(* Logix 5000 project; controller STAT 1756-L72 rev 20.12; software revision 20.04; part 25 of 34 *)
(* tags used below, declared in another part *)
   B3 : DINT[35];
   N7 : DINT[150];
   N9 : DINT[200];
   S : INT[164];
   T4 : TIMER[100];
   tempo_d_lvl_H_decL1 : TIMER;
   tempo_on_lvl_H_decL1 : TIMER;
(* LANCY, continued *)

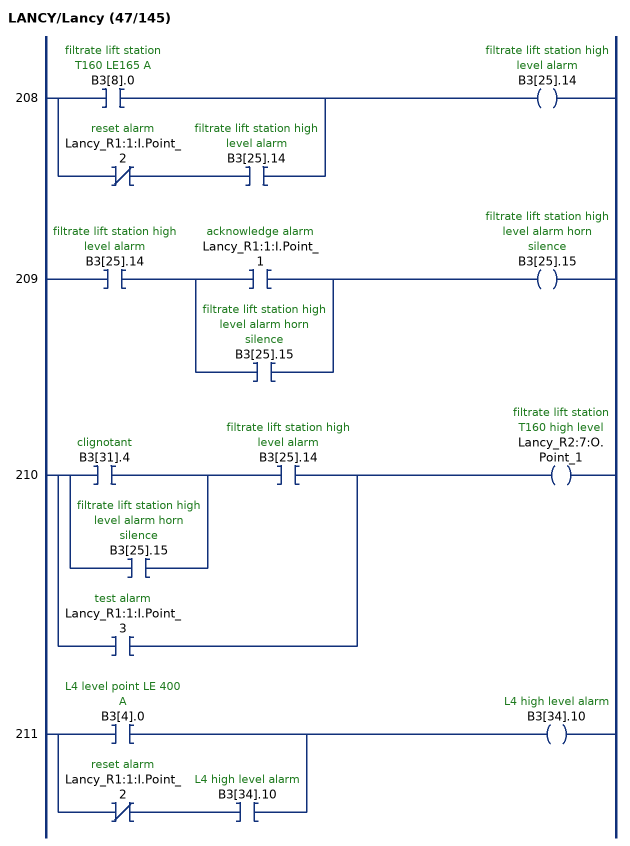
   208: [XIC(B3[8].0) ,XIO(Lancy_R1:1:I.Point_2) XIC(B3[25].14) ]OTE(B3[25].14);
   209: XIC(B3[25].14)[XIC(Lancy_R1:1:I.Point_1) ,XIC(B3[25].15) ]OTE(B3[25].15);
   210: [[XIC(B3[31].4) ,XIC(B3[25].15) ] XIC(B3[25].14) ,XIC(Lancy_R1:1:I.Point_3) ]OTE(Lancy_R2:7:O.Point_1);
   211: [XIC(B3[4].0) ,XIO(Lancy_R1:1:I.Point_2) XIC(B3[34].10) ]OTE(B3[34].10);
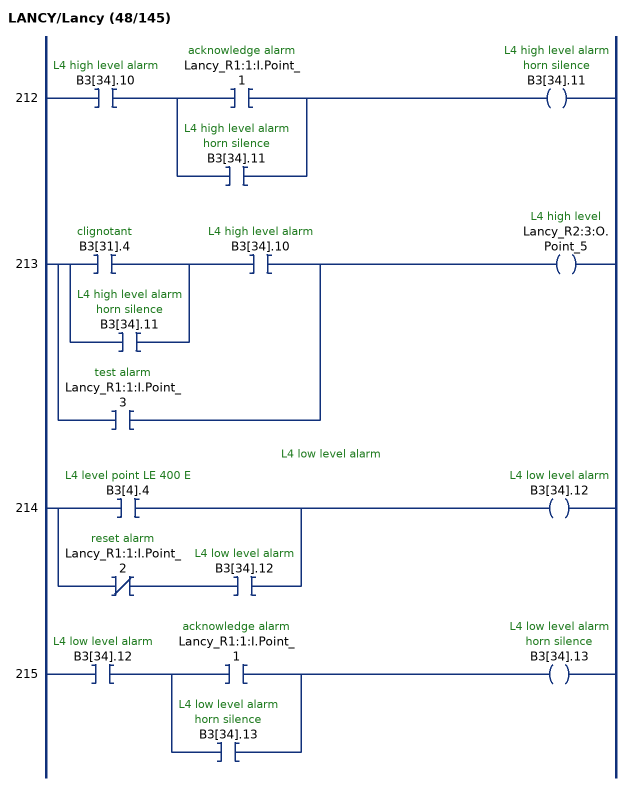
   212: XIC(B3[34].10)[XIC(Lancy_R1:1:I.Point_1) ,XIC(B3[34].11) ]OTE(B3[34].11);
   213: [[XIC(B3[31].4) ,XIC(B3[34].11) ] XIC(B3[34].10) ,XIC(Lancy_R1:1:I.Point_3) ]OTE(Lancy_R2:3:O.Point_5);
   // L4 low level alarm
   214: [XIC(B3[4].4) ,XIO(Lancy_R1:1:I.Point_2) XIC(B3[34].12) ]OTE(B3[34].12);
   215: XIC(B3[34].12)[XIC(Lancy_R1:1:I.Point_1) ,XIC(B3[34].13) ]OTE(B3[34].13);
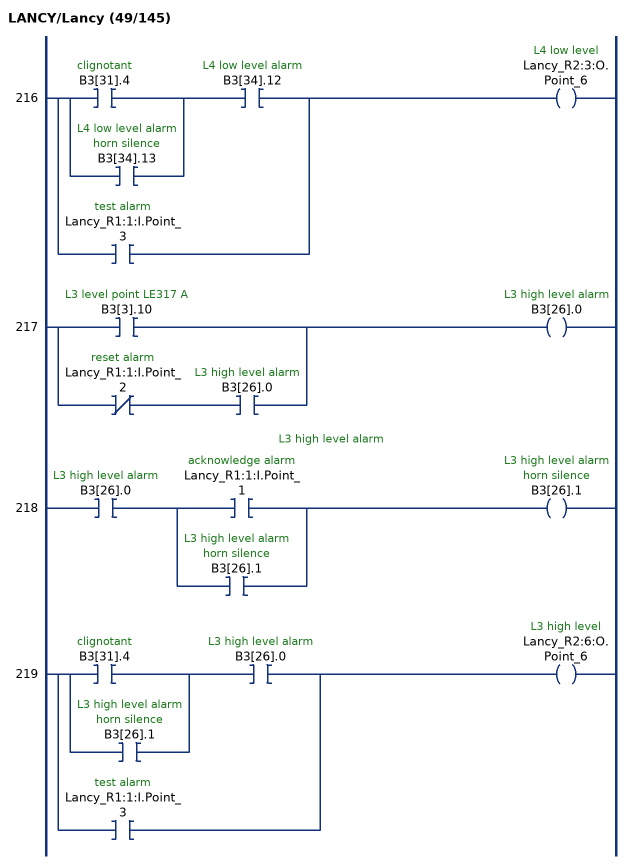
   216: [[XIC(B3[31].4) ,XIC(B3[34].13) ] XIC(B3[34].12) ,XIC(Lancy_R1:1:I.Point_3) ]OTE(Lancy_R2:3:O.Point_6);
   217: [XIC(B3[3].10) ,XIO(Lancy_R1:1:I.Point_2) XIC(B3[26].0) ]OTE(B3[26].0);
   // L3 high level alarm
   218: XIC(B3[26].0)[XIC(Lancy_R1:1:I.Point_1) ,XIC(B3[26].1) ]OTE(B3[26].1);
   219: [[XIC(B3[31].4) ,XIC(B3[26].1) ] XIC(B3[26].0) ,XIC(Lancy_R1:1:I.Point_3) ]OTE(Lancy_R2:6:O.Point_6);
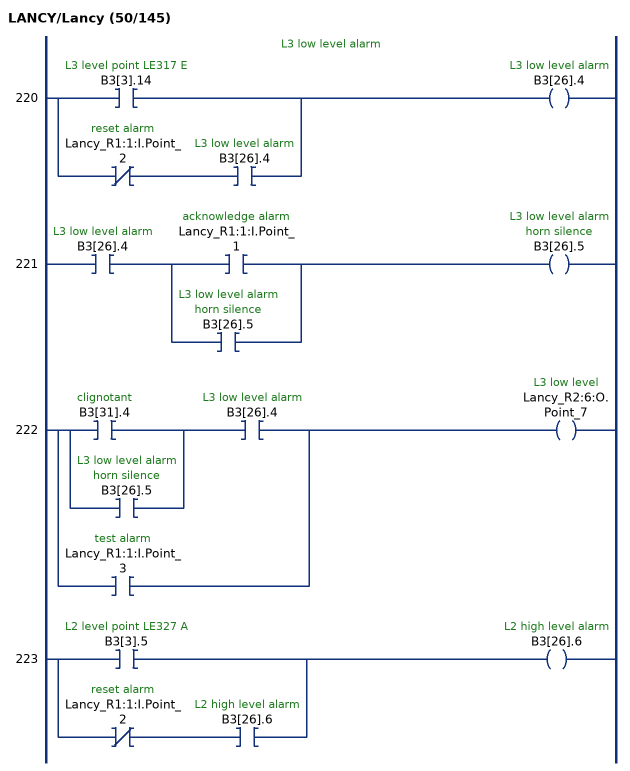
   // L3 low level alarm
   220: [XIC(B3[3].14) ,XIO(Lancy_R1:1:I.Point_2) XIC(B3[26].4) ]OTE(B3[26].4);
   221: XIC(B3[26].4)[XIC(Lancy_R1:1:I.Point_1) ,XIC(B3[26].5) ]OTE(B3[26].5);
   222: [[XIC(B3[31].4) ,XIC(B3[26].5) ] XIC(B3[26].4) ,XIC(Lancy_R1:1:I.Point_3) ]OTE(Lancy_R2:6:O.Point_7);
   223: [XIC(B3[3].5) ,XIO(Lancy_R1:1:I.Point_2) XIC(B3[26].6) ]OTE(B3[26].6);
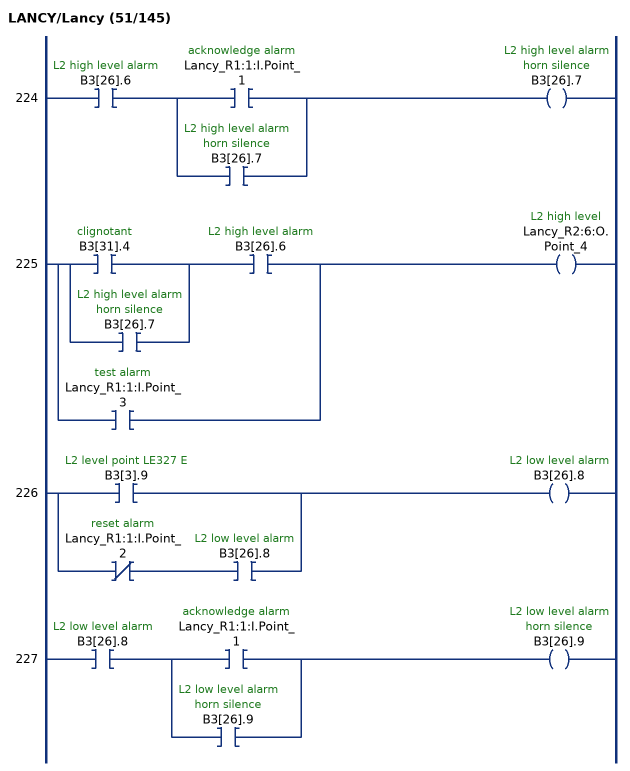
   224: XIC(B3[26].6)[XIC(Lancy_R1:1:I.Point_1) ,XIC(B3[26].7) ]OTE(B3[26].7);
   225: [[XIC(B3[31].4) ,XIC(B3[26].7) ] XIC(B3[26].6) ,XIC(Lancy_R1:1:I.Point_3) ]OTE(Lancy_R2:6:O.Point_4);
   226: [XIC(B3[3].9) ,XIO(Lancy_R1:1:I.Point_2) XIC(B3[26].8) ]OTE(B3[26].8);
   227: XIC(B3[26].8)[XIC(Lancy_R1:1:I.Point_1) ,XIC(B3[26].9) ]OTE(B3[26].9);
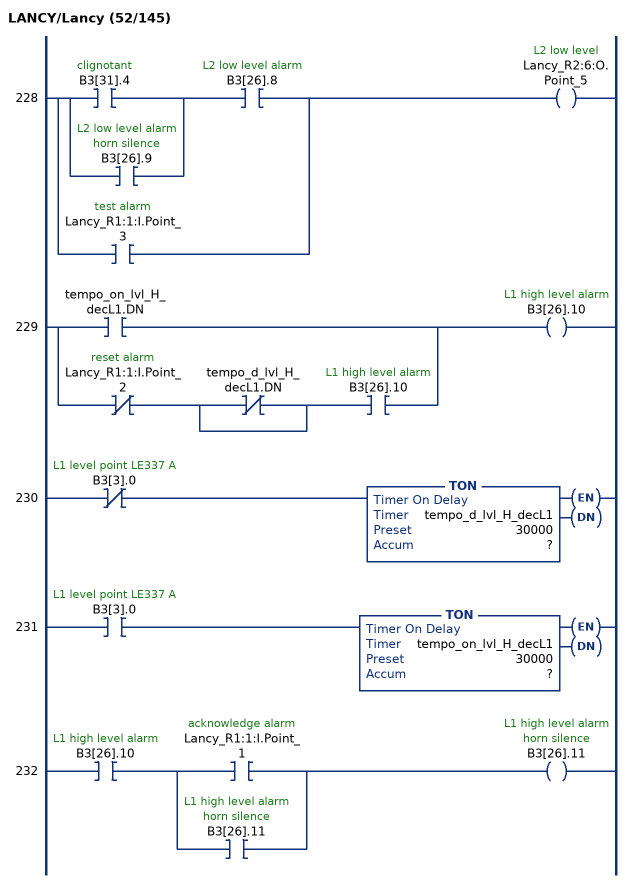
   228: [[XIC(B3[31].4) ,XIC(B3[26].9) ] XIC(B3[26].8) ,XIC(Lancy_R1:1:I.Point_3) ]OTE(Lancy_R2:6:O.Point_5);
   229: [XIC(tempo_on_lvl_H_decL1.DN) ,XIO(Lancy_R1:1:I.Point_2) [XIO(tempo_d_lvl_H_decL1.DN) ,] XIC(B3[26].10) ]OTE(B3[26].10);
   230: XIO(B3[3].0)TON(tempo_d_lvl_H_decL1,?,?);
   231: XIC(B3[3].0)TON(tempo_on_lvl_H_decL1,?,?);
   232: XIC(B3[26].10)[XIC(Lancy_R1:1:I.Point_1) ,XIC(B3[26].11) ]OTE(B3[26].11);
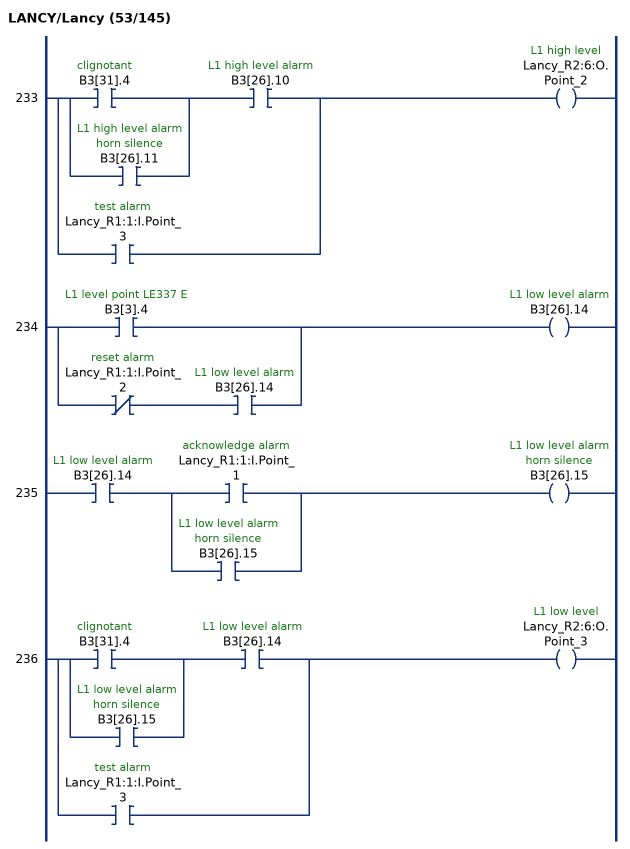
   233: [[XIC(B3[31].4) ,XIC(B3[26].11) ] XIC(B3[26].10) ,XIC(Lancy_R1:1:I.Point_3) ]OTE(Lancy_R2:6:O.Point_2);
   234: [XIC(B3[3].4) ,XIO(Lancy_R1:1:I.Point_2) XIC(B3[26].14) ]OTE(B3[26].14);
   235: XIC(B3[26].14)[XIC(Lancy_R1:1:I.Point_1) ,XIC(B3[26].15) ]OTE(B3[26].15);
   236: [[XIC(B3[31].4) ,XIC(B3[26].15) ] XIC(B3[26].14) ,XIC(Lancy_R1:1:I.Point_3) ]OTE(Lancy_R2:6:O.Point_3);
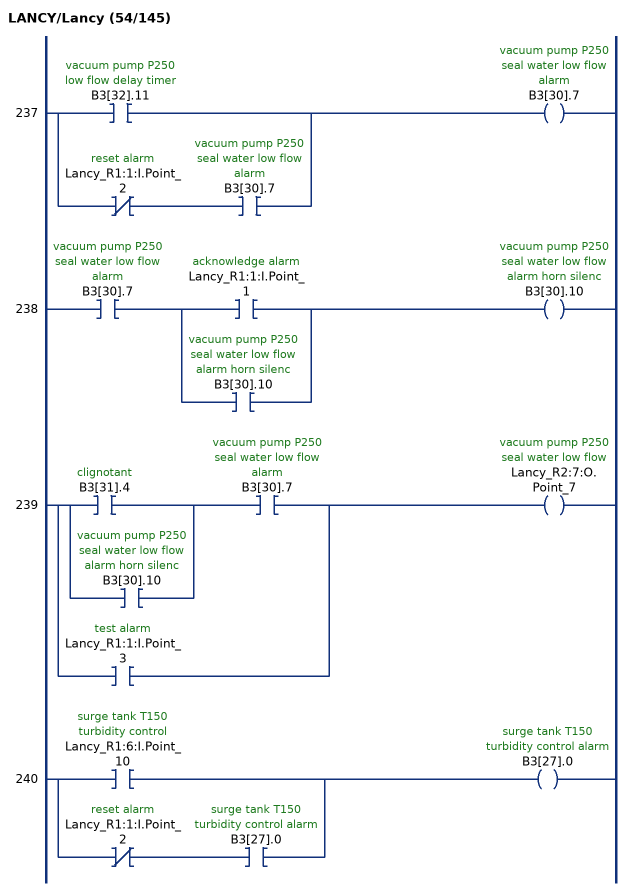
   237: [XIC(B3[32].11) ,XIO(Lancy_R1:1:I.Point_2) XIC(B3[30].7) ]OTE(B3[30].7);
   238: XIC(B3[30].7)[XIC(Lancy_R1:1:I.Point_1) ,XIC(B3[30].10) ]OTE(B3[30].10);
   239: [[XIC(B3[31].4) ,XIC(B3[30].10) ] XIC(B3[30].7) ,XIC(Lancy_R1:1:I.Point_3) ]OTE(Lancy_R2:7:O.Point_7);
   240: [XIC(Lancy_R1:6:I.Point_10) ,XIO(Lancy_R1:1:I.Point_2) XIC(B3[27].0) ]OTE(B3[27].0);
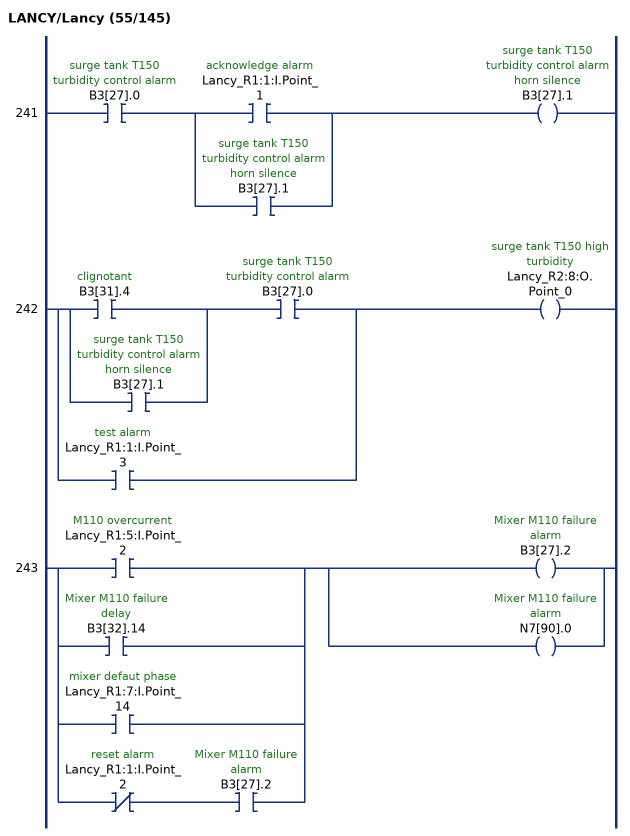
   241: XIC(B3[27].0)[XIC(Lancy_R1:1:I.Point_1) ,XIC(B3[27].1) ]OTE(B3[27].1);
   242: [[XIC(B3[31].4) ,XIC(B3[27].1) ] XIC(B3[27].0) ,XIC(Lancy_R1:1:I.Point_3) ]OTE(Lancy_R2:8:O.Point_0);
   243: [[XIC(Lancy_R1:5:I.Point_2) ,XIC(B3[32].14) ,XIC(Lancy_R1:7:I.Point_14) ] ,XIO(Lancy_R1:1:I.Point_2) XIC(B3[27].2) ][OTE(B3[27].2) ,OTE(N7[90].0) ];
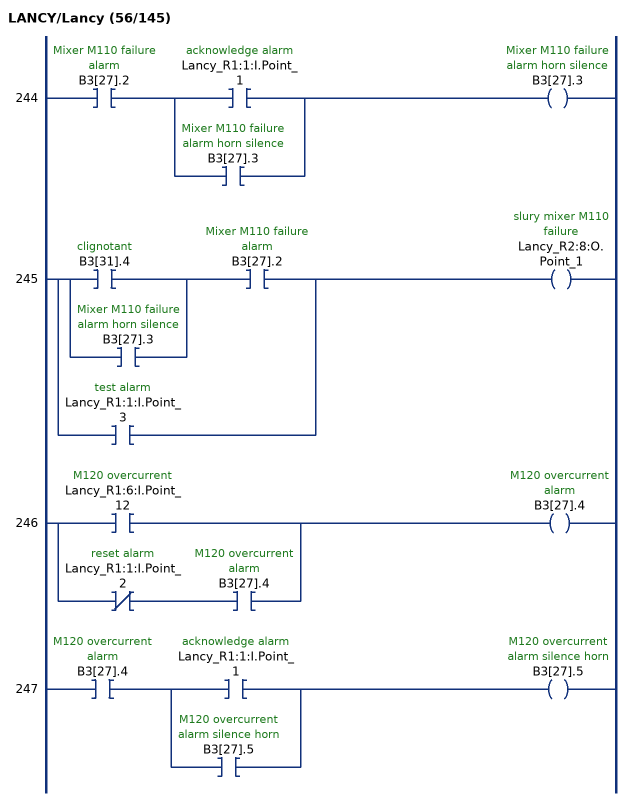
   244: XIC(B3[27].2)[XIC(Lancy_R1:1:I.Point_1) ,XIC(B3[27].3) ]OTE(B3[27].3);
   245: [[XIC(B3[31].4) ,XIC(B3[27].3) ] XIC(B3[27].2) ,XIC(Lancy_R1:1:I.Point_3) ]OTE(Lancy_R2:8:O.Point_1);
   246: [XIC(Lancy_R1:6:I.Point_12) ,XIO(Lancy_R1:1:I.Point_2) XIC(B3[27].4) ]OTE(B3[27].4);
   247: XIC(B3[27].4)[XIC(Lancy_R1:1:I.Point_1) ,XIC(B3[27].5) ]OTE(B3[27].5);
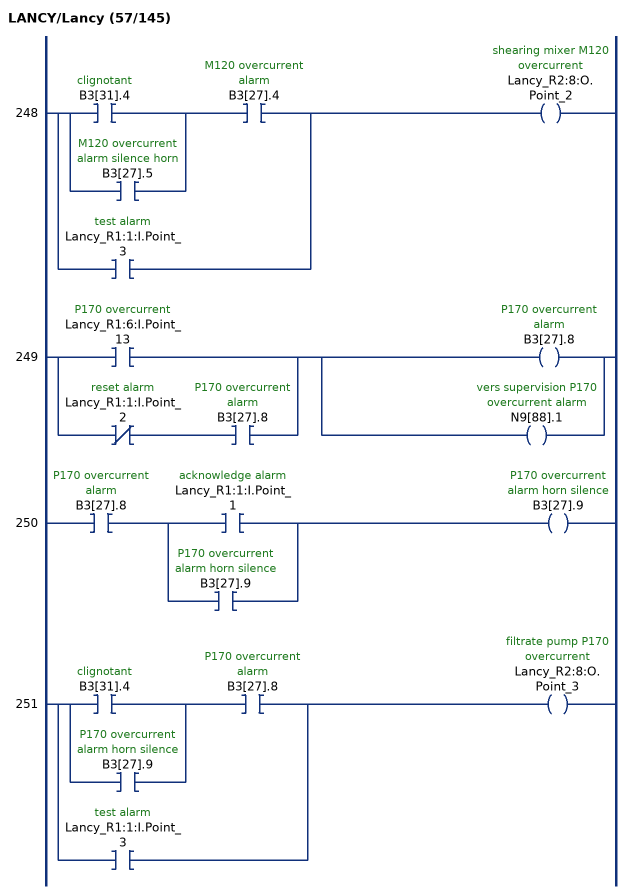
   248: [[XIC(B3[31].4) ,XIC(B3[27].5) ] XIC(B3[27].4) ,XIC(Lancy_R1:1:I.Point_3) ]OTE(Lancy_R2:8:O.Point_2);
   249: [XIC(Lancy_R1:6:I.Point_13) ,XIO(Lancy_R1:1:I.Point_2) XIC(B3[27].8) ][OTE(B3[27].8) ,OTE(N9[88].1) ];
   250: XIC(B3[27].8)[XIC(Lancy_R1:1:I.Point_1) ,XIC(B3[27].9) ]OTE(B3[27].9);
   251: [[XIC(B3[31].4) ,XIC(B3[27].9) ] XIC(B3[27].8) ,XIC(Lancy_R1:1:I.Point_3) ]OTE(Lancy_R2:8:O.Point_3);
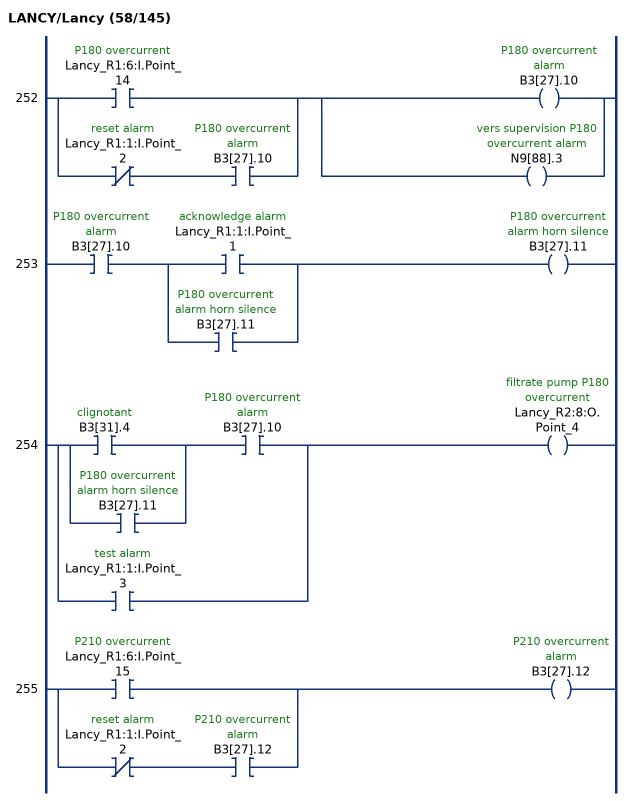
   252: [XIC(Lancy_R1:6:I.Point_14) ,XIO(Lancy_R1:1:I.Point_2) XIC(B3[27].10) ][OTE(B3[27].10) ,OTE(N9[88].3) ];
   253: XIC(B3[27].10)[XIC(Lancy_R1:1:I.Point_1) ,XIC(B3[27].11) ]OTE(B3[27].11);
   254: [[XIC(B3[31].4) ,XIC(B3[27].11) ] XIC(B3[27].10) ,XIC(Lancy_R1:1:I.Point_3) ]OTE(Lancy_R2:8:O.Point_4);
   255: [XIC(Lancy_R1:6:I.Point_15) ,XIO(Lancy_R1:1:I.Point_2) XIC(B3[27].12) ]OTE(B3[27].12);
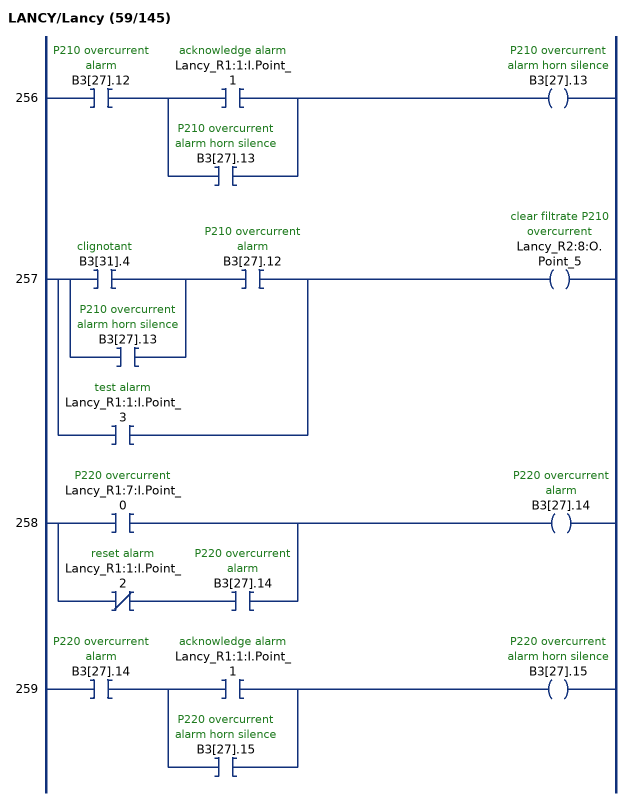
   256: XIC(B3[27].12)[XIC(Lancy_R1:1:I.Point_1) ,XIC(B3[27].13) ]OTE(B3[27].13);
   257: [[XIC(B3[31].4) ,XIC(B3[27].13) ] XIC(B3[27].12) ,XIC(Lancy_R1:1:I.Point_3) ]OTE(Lancy_R2:8:O.Point_5);
   258: [XIC(Lancy_R1:7:I.Point_0) ,XIO(Lancy_R1:1:I.Point_2) XIC(B3[27].14) ]OTE(B3[27].14);
   259: XIC(B3[27].14)[XIC(Lancy_R1:1:I.Point_1) ,XIC(B3[27].15) ]OTE(B3[27].15);
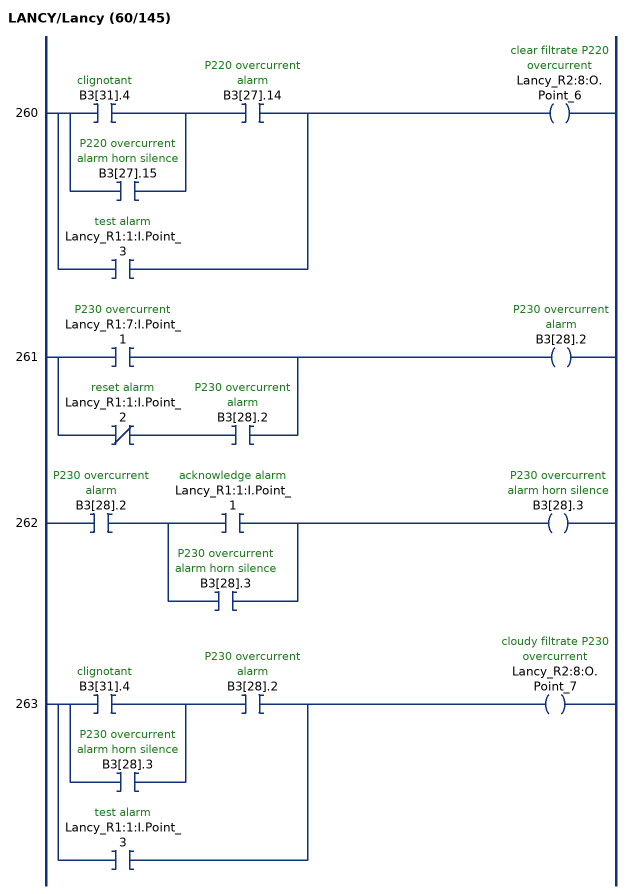
   260: [[XIC(B3[31].4) ,XIC(B3[27].15) ] XIC(B3[27].14) ,XIC(Lancy_R1:1:I.Point_3) ]OTE(Lancy_R2:8:O.Point_6);
   261: [XIC(Lancy_R1:7:I.Point_1) ,XIO(Lancy_R1:1:I.Point_2) XIC(B3[28].2) ]OTE(B3[28].2);
   262: XIC(B3[28].2)[XIC(Lancy_R1:1:I.Point_1) ,XIC(B3[28].3) ]OTE(B3[28].3);
   263: [[XIC(B3[31].4) ,XIC(B3[28].3) ] XIC(B3[28].2) ,XIC(Lancy_R1:1:I.Point_3) ]OTE(Lancy_R2:8:O.Point_7);
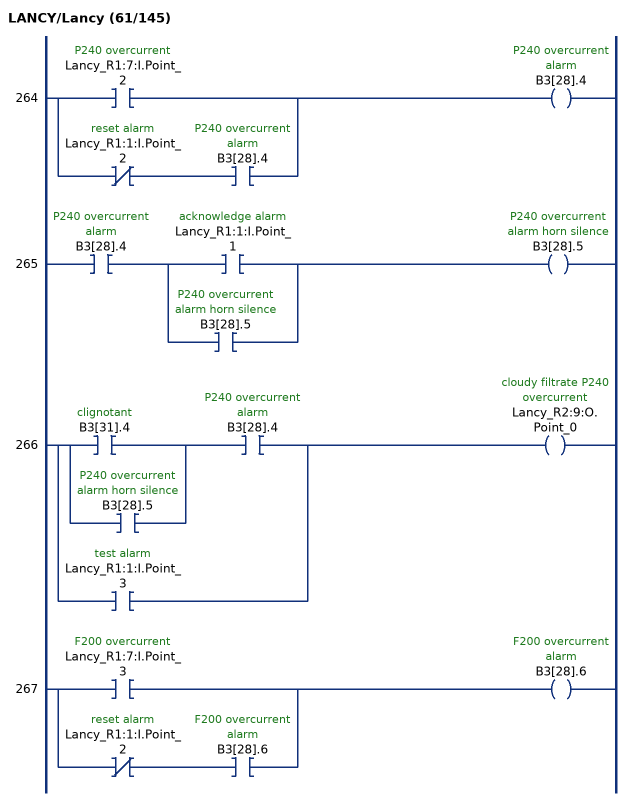
   264: [XIC(Lancy_R1:7:I.Point_2) ,XIO(Lancy_R1:1:I.Point_2) XIC(B3[28].4) ]OTE(B3[28].4);
   265: XIC(B3[28].4)[XIC(Lancy_R1:1:I.Point_1) ,XIC(B3[28].5) ]OTE(B3[28].5);
   266: [[XIC(B3[31].4) ,XIC(B3[28].5) ] XIC(B3[28].4) ,XIC(Lancy_R1:1:I.Point_3) ]OTE(Lancy_R2:9:O.Point_0);
   267: [XIC(Lancy_R1:7:I.Point_3) ,XIO(Lancy_R1:1:I.Point_2) XIC(B3[28].6) ]OTE(B3[28].6);
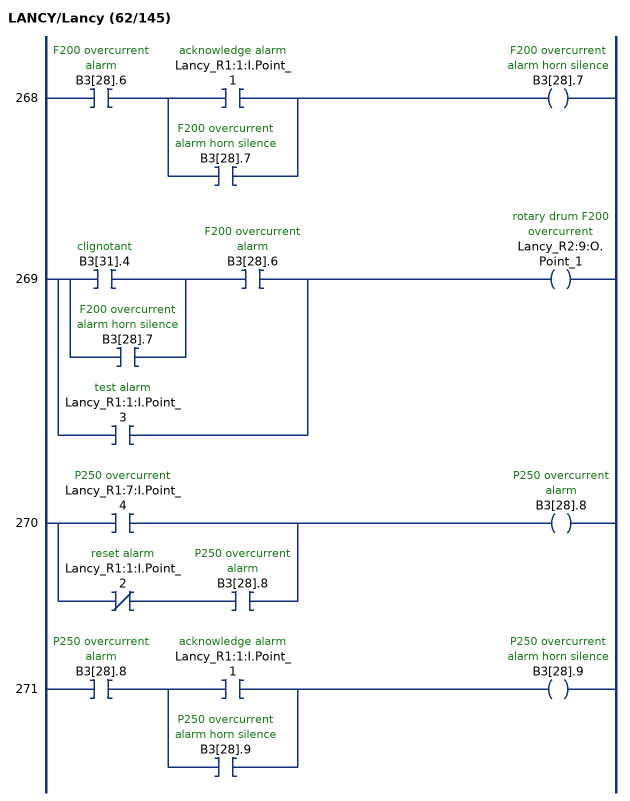
   268: XIC(B3[28].6)[XIC(Lancy_R1:1:I.Point_1) ,XIC(B3[28].7) ]OTE(B3[28].7);
   269: [[XIC(B3[31].4) ,XIC(B3[28].7) ] XIC(B3[28].6) ,XIC(Lancy_R1:1:I.Point_3) ]OTE(Lancy_R2:9:O.Point_1);
   270: [XIC(Lancy_R1:7:I.Point_4) ,XIO(Lancy_R1:1:I.Point_2) XIC(B3[28].8) ]OTE(B3[28].8);
   271: XIC(B3[28].8)[XIC(Lancy_R1:1:I.Point_1) ,XIC(B3[28].9) ]OTE(B3[28].9);
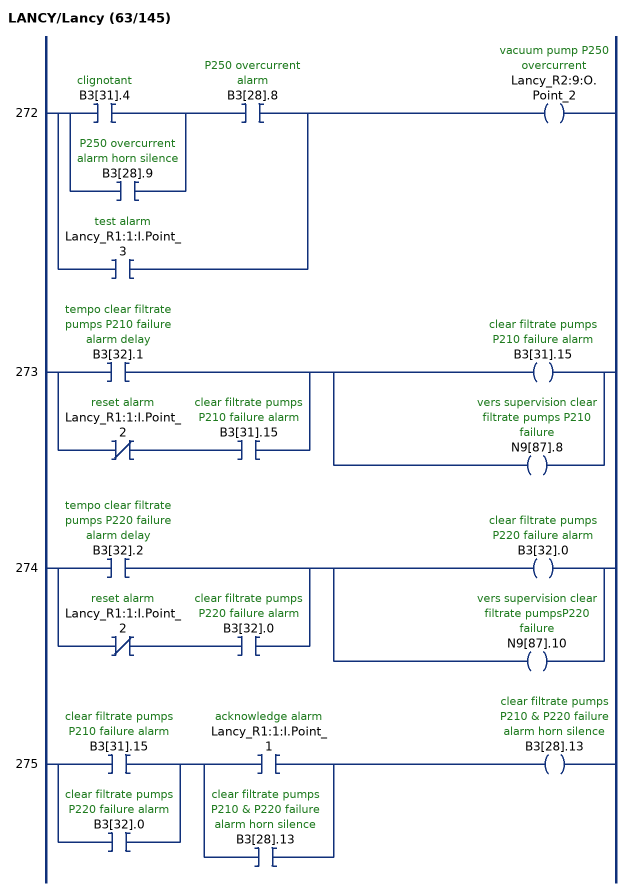
   272: [[XIC(B3[31].4) ,XIC(B3[28].9) ] XIC(B3[28].8) ,XIC(Lancy_R1:1:I.Point_3) ]OTE(Lancy_R2:9:O.Point_2);
   273: [XIC(B3[32].1) ,XIO(Lancy_R1:1:I.Point_2) XIC(B3[31].15) ][OTE(B3[31].15) ,OTE(N9[87].8) ];
   274: [XIC(B3[32].2) ,XIO(Lancy_R1:1:I.Point_2) XIC(B3[32].0) ][OTE(B3[32].0) ,OTE(N9[87].10) ];
   275: [XIC(B3[31].15) ,XIC(B3[32].0) ][XIC(Lancy_R1:1:I.Point_1) ,XIC(B3[28].13) ]OTE(B3[28].13);
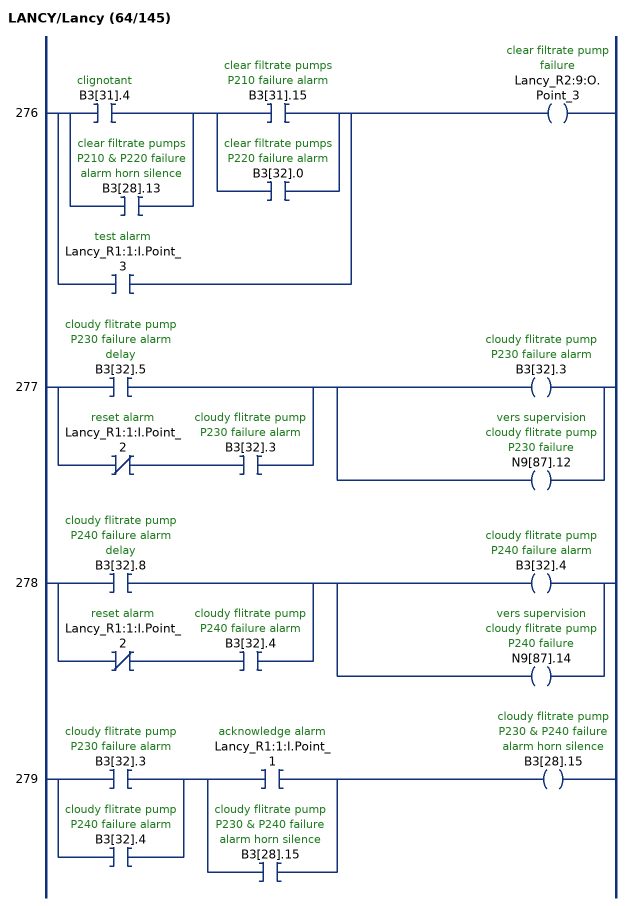
   276: [[XIC(B3[31].4) ,XIC(B3[28].13) ] [XIC(B3[31].15) ,XIC(B3[32].0) ] ,XIC(Lancy_R1:1:I.Point_3) ]OTE(Lancy_R2:9:O.Point_3);
   277: [XIC(B3[32].5) ,XIO(Lancy_R1:1:I.Point_2) XIC(B3[32].3) ][OTE(B3[32].3) ,OTE(N9[87].12) ];
   278: [XIC(B3[32].8) ,XIO(Lancy_R1:1:I.Point_2) XIC(B3[32].4) ][OTE(B3[32].4) ,OTE(N9[87].14) ];
   279: [XIC(B3[32].3) ,XIC(B3[32].4) ][XIC(Lancy_R1:1:I.Point_1) ,XIC(B3[28].15) ]OTE(B3[28].15);
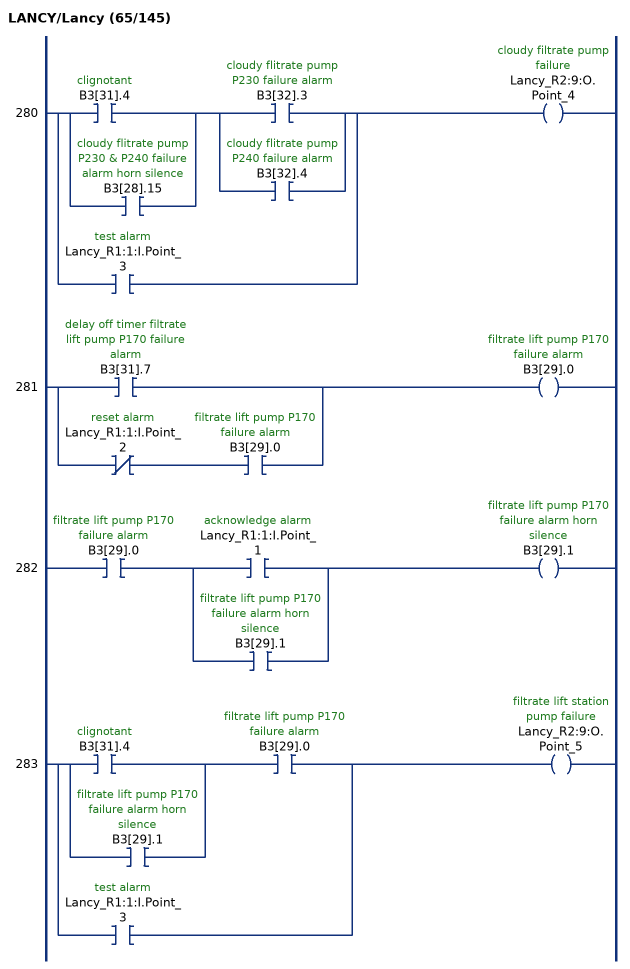
   280: [[XIC(B3[31].4) ,XIC(B3[28].15) ] [XIC(B3[32].3) ,XIC(B3[32].4) ] ,XIC(Lancy_R1:1:I.Point_3) ]OTE(Lancy_R2:9:O.Point_4);
   281: [XIC(B3[31].7) ,XIO(Lancy_R1:1:I.Point_2) XIC(B3[29].0) ]OTE(B3[29].0);
   282: XIC(B3[29].0)[XIC(Lancy_R1:1:I.Point_1) ,XIC(B3[29].1) ]OTE(B3[29].1);
   283: [[XIC(B3[31].4) ,XIC(B3[29].1) ] XIC(B3[29].0) ,XIC(Lancy_R1:1:I.Point_3) ]OTE(Lancy_R2:9:O.Point_5);
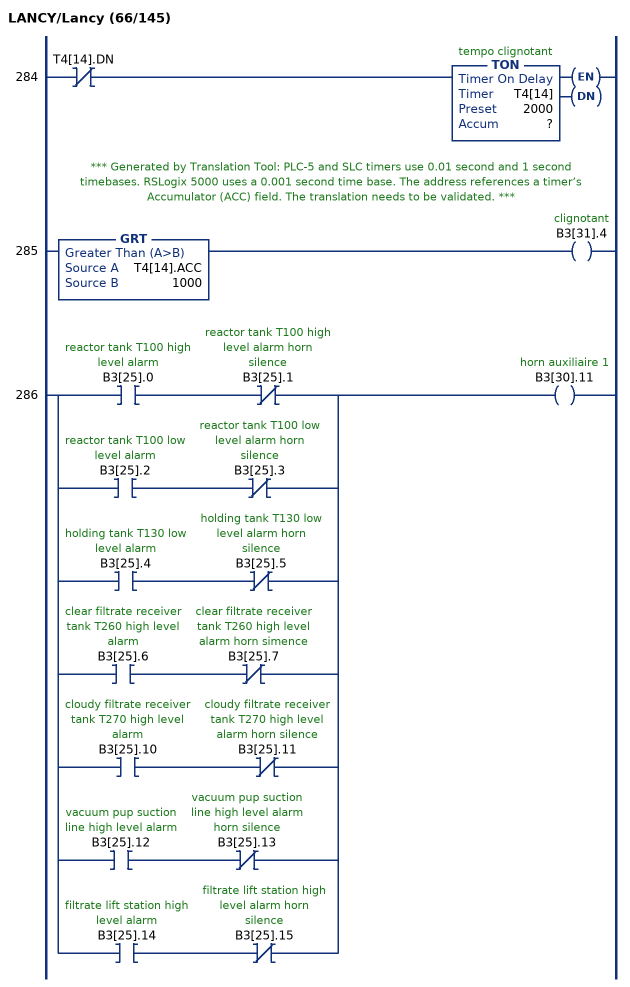
   284: XIO(T4[14].DN)TON(T4[14],?,?);
   // *** Generated by Translation Tool: PLC-5 and SLC timers use 0.01 second and 1 second timebases. RSLogix 5000 uses a 0.001 second time base. The address references a timer’s Accumulator (ACC) field. The translation needs to be validated. ***
   285: GRT(T4[14].ACC,1000)OTE(B3[31].4);
   286: [XIC(B3[25].0) XIO(B3[25].1) ,XIC(B3[25].2) XIO(B3[25].3) ,XIC(B3[25].4) XIO(B3[25].5) ,XIC(B3[25].6) XIO(B3[25].7) ,XIC(B3[25].10) XIO(B3[25].11) ,XIC(B3[25].12) XIO(B3[25].13) ,XIC(B3[25].14) XIO(B3[25].15) ]OTE(B3[30].11);
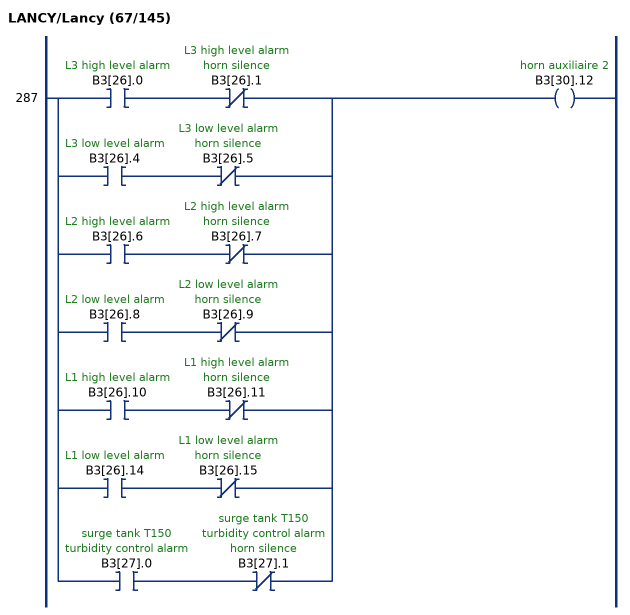
   287: [XIC(B3[26].0) XIO(B3[26].1) ,XIC(B3[26].4) XIO(B3[26].5) ,XIC(B3[26].6) XIO(B3[26].7) ,XIC(B3[26].8) XIO(B3[26].9) ,XIC(B3[26].10) XIO(B3[26].11) ,XIC(B3[26].14) XIO(B3[26].15) ,XIC(B3[27].0) XIO(B3[27].1) ]OTE(B3[30].12);
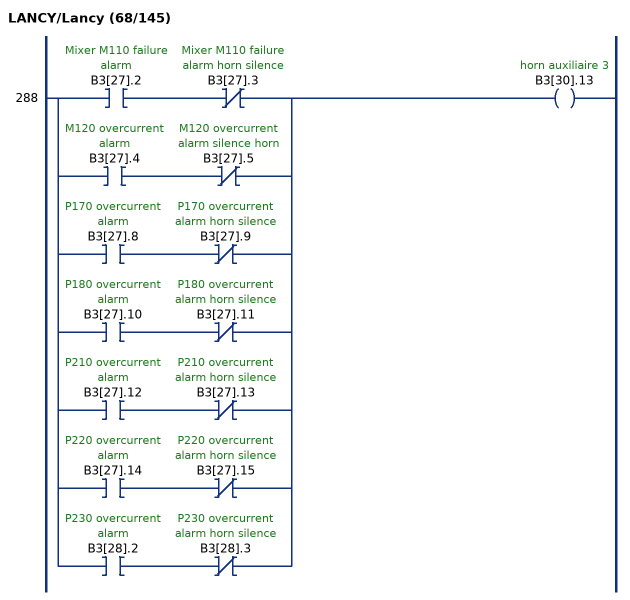
   288: [XIC(B3[27].2) XIO(B3[27].3) ,XIC(B3[27].4) XIO(B3[27].5) ,XIC(B3[27].8) XIO(B3[27].9) ,XIC(B3[27].10) XIO(B3[27].11) ,XIC(B3[27].12) XIO(B3[27].13) ,XIC(B3[27].14) XIO(B3[27].15) ,XIC(B3[28].2) XIO(B3[28].3) ]OTE(B3[30].13);
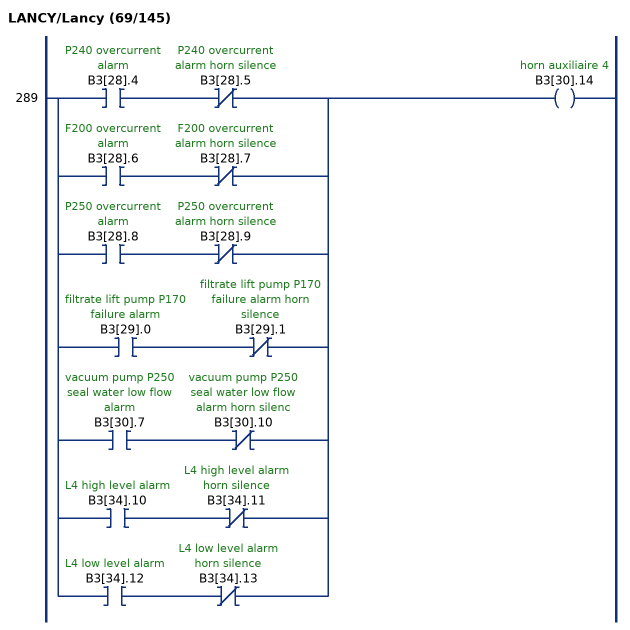
   289: [XIC(B3[28].4) XIO(B3[28].5) ,XIC(B3[28].6) XIO(B3[28].7) ,XIC(B3[28].8) XIO(B3[28].9) ,XIC(B3[29].0) XIO(B3[29].1) ,XIC(B3[30].7) XIO(B3[30].10) ,XIC(B3[34].10) XIO(B3[34].11) ,XIC(B3[34].12) XIO(B3[34].13) ]OTE(B3[30].14);
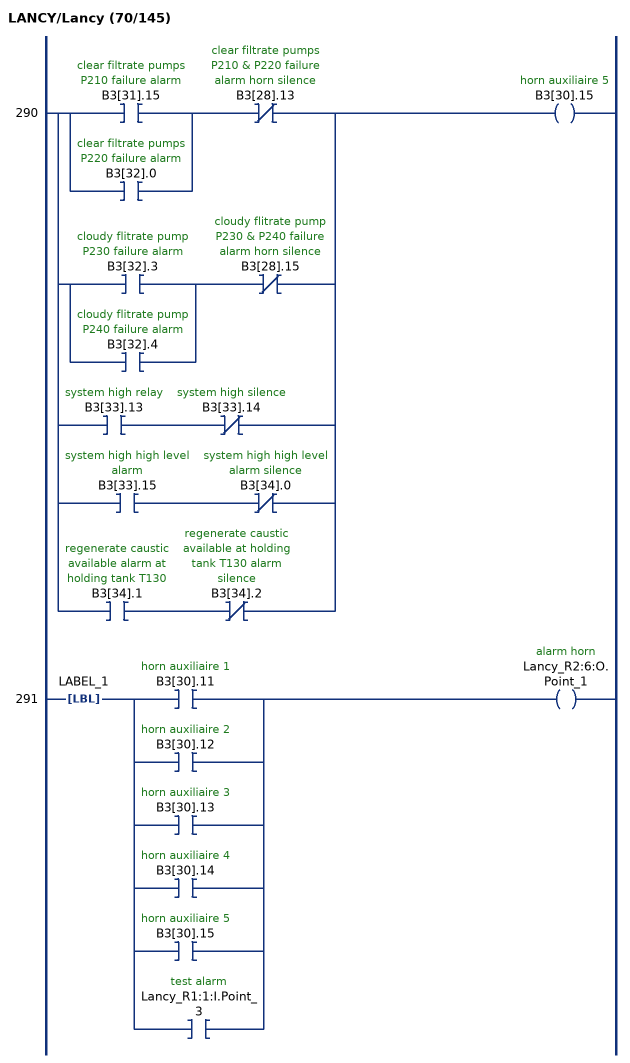
   290: [[XIC(B3[31].15) ,XIC(B3[32].0) ] XIO(B3[28].13) ,[XIC(B3[32].3) ,XIC(B3[32].4) ] XIO(B3[28].15) ,XIC(B3[33].13) XIO(B3[33].14) ,XIC(B3[33].15) XIO(B3[34].0) ,XIC(B3[34].1) XIO(B3[34].2) ]OTE(B3[30].15);
   291: LBL(LABEL_1)[XIC(B3[30].11) ,XIC(B3[30].12) ,XIC(B3[30].13) ,XIC(B3[30].14) ,XIC(B3[30].15) ,XIC(Lancy_R1:1:I.Point_3) ]OTE(Lancy_R2:6:O.Point_1);
